{attribute addProperty BoxType "KL3361-0001"}
{attribute addProperty Id "Channel_1Channel_C961C78600"}
{attribute addProperty CRC "3532189323"}
{attribute addProperty SizeInBites "0"}
{attribute addProperty SizeInBytes "0"}
TYPE KL_D288EE8B :
STRUCT
	{attribute addProperty Name "Channel_1"}
	Channel_1 : Channel_C961C786;
END_STRUCT
END_TYPE

(* stored: Version 1.2.0.0, ProductVersion 3.1.4024.9
   DUT KL_D288EE8B: Id {05a238e2-47f1-439b-8741-fbd02b50511d} *)
